FUNCTION RAD2DEGRE : lreal
VAR_INPUT
	lrAngle : LREAL;
END_VAR
VAR
END_VAR

RAD2DEGRE := lrAngle*180/PI;

END_FUNCTION

(* stored: Version 1.1.0.1, ProductVersion 3.1.4024.11
   POU RAD2DEGRE: Id {5756c9d0-4f43-4713-939f-ec4e279302a2}, SpecialFunc None *)
